FUNCTION_BLOCK FB_CH_Object IMPLEMENTS I_CH_Object
VAR
	fbSourceInfo : FB_TcSourceInfo;
	
	{attribute 'hide'}
	nTaskIndex : BYTE; //Used in TwinCAT_SystemInfoVarList._TaskInfo
END_VAR

METHOD FB_init : BOOL
VAR_INPUT
	bInitRetains : BOOL; // if TRUE, the retain variables are initialized (warm start / cold start)
	bInCopyCode : BOOL;  // if TRUE, the instance afterwards gets moved into the copy code (online change)
END_VAR
VAR
	fbGetCurTaskIdx  : GETCURTASKINDEX;
END_VAR
fbGetCurTaskIdx();
THIS^.nTaskIndex := fbGetCurTaskIdx.Index;
END_METHOD

METHOD Initialize : HRESULT
Initialize := S_OK;
END_METHOD

{attribute 'monitoring':='call'}
PROPERTY LUID : STRING //Locally unique identifier
GET
LUID := THIS^.fbSourceInfo.sName;
END_GET
END_PROPERTY

{attribute 'monitoring':='call'}
PROPERTY OID : OTCID //Object ID
GET
OID := 0;
END_GET
END_PROPERTY

PROPERTY PROTECTED TaskIndex : BYTE //Used in TwinCAT_SystemInfoVarList._TaskInfo
GET
TaskIndex := THIS^.nTaskIndex;
END_GET
END_PROPERTY

METHOD Update : HRESULT
VAR_INPUT
END_VAR
Update := S_OK;
END_METHOD

END_FUNCTION_BLOCK

(* stored: Version 1.1.0.1, ProductVersion 3.1.4024.12
   POU FB_CH_Object: Id {409d828e-23b5-4a9e-a56a-5036375242c4}, SpecialFunc None
   Method FB_init: Id {0fae9e54-ec66-40c1-b480-f848bab32e25}
   Method Initialize: Id {be8a023b-6296-4807-8e60-e5a7f80de0fd}
   Property LUID: Id {474686ea-ffab-47fd-a05b-420d3e45ce29}
   Get Get: Id {c098fcbe-8b71-42a1-b28d-abed1ec65b4b}
   Property OID: Id {e3dde703-13aa-48d9-895b-2f28dd4ec172}
   Get Get: Id {3291e80a-1091-4808-a53b-7a3c33206193}
   Property TaskIndex: Id {0d71e8a5-11e0-4564-a8a9-71aaa9db2e92}
   Get Get: Id {5482258d-f630-44e1-8f58-c8cf236fbd5d}
   Method Update: Id {803c0f33-543c-4185-9957-af53704b5468} *)
